// TwinCAT 3 PLC project plc01
// ProgramVersion: 3.1.4026.20
// libraries:
//   Tc2_Standard, * (Beckhoff Automation GmbH)
//   Tc2_System, * (Beckhoff Automation GmbH)
//   Tc2_Utilities, * (Beckhoff Automation GmbH)
//   Tc3_Event, * (www.peterzerlauth.com)
// project tree:
//   / FastTask.TcTTO (not stored), PlcTask.TcTTO (not stored)
//   POUs/ FAST.TcPOU (not stored), FB_TestSlow.TcPOU, FB_TestFast.TcPOU, MAIN.TcPOU
// real-time tasks:
//   TASK SlowTask: cycle T#20ms, priority 20, ADS port 350
//   TASK FastTask: cycle T#1ms, priority 1, ADS port 351

// ---- POUs/FB_TestSlow.TcPOU
FUNCTION_BLOCK FB_TestSlow
VAR_INPUT
END_VAR
VAR_OUTPUT
END_VAR
VAR
	fbEvent: 			Tc3_Event.FB_Event;
	bVerbose:			BOOL;
	bInfo:				BOOL;
	bWarning:			BOOL;
	bError:				BOOL;
	bCritical:			BOOL;

END_VAR

fbEvent();

// Demonstration of FB_Event usage with various log levels and argument types

IF bVerbose THEN
	fbEvent.P_Argument.M_AddINT(134052566194980000);
	fbEvent.P_Argument.M_AddSTRING('mm');
	fbEvent.M_Verbose('V message %s %s');
END_IF

IF bInfo THEN
	fbEvent.P_Argument.M_AddREAL(33.134581234, 3);
	fbEvent.P_Argument.M_AddSTRING('mm');
	fbEvent.M_Info('I message %s %s', 0);
END_IF

IF bWarning THEN
	fbEvent.M_Warning('W message', 0);
	fbEvent.M_Warning('B message', 475719253);
END_IF

IF bError THEN
	fbEvent.M_Error('E message', 475719235);
END_IF

IF bCritical THEN
	fbEvent.M_Error('Input %s is simulated', 849363082);
END_IF

PROPERTY PUBLIC P_Event : reference to FB_event
GET
P_Event ref= fbEvent;
END_GET
END_PROPERTY

END_FUNCTION_BLOCK

// ---- POUs/FB_TestFast.TcPOU
FUNCTION_BLOCK FB_TestFast
VAR_INPUT
END_VAR
VAR_OUTPUT
END_VAR
VAR
	fbEvent: 			Tc3_Event.FB_Event;
	bVerbose:			BOOL;
	bInfo:				BOOL;
	bWarning:			BOOL;
	bError:				BOOL;
	bCritical:			BOOL;

END_VAR

fbEvent();

// Demonstration of FB_Event usage with various log levels and argument types

IF bVerbose THEN
	fbEvent.P_Argument.M_AddINT(134052566194980000);
	fbEvent.P_Argument.M_AddSTRING('mm');
	fbEvent.M_Verbose('V message %s %s');
END_IF

IF bInfo THEN
	fbEvent.P_Argument.M_AddREAL(33.134581234, 3);
	fbEvent.P_Argument.M_AddSTRING('mm');
	fbEvent.M_Info('I message %s %s', 828536003);
END_IF

IF bWarning THEN
	fbEvent.M_Warning('W message', 475719253);
	fbEvent.M_Warning('W message', 475719253);
END_IF

IF bError THEN
	fbEvent.M_Error('E message', 475719235);
END_IF

IF bCritical THEN
	fbEvent.M_Critical('C message', 475719233); ///839384782
	fbEvent.M_Critical('B message', 0); 
END_IF

PROPERTY PUBLIC P_Event : reference to FB_event
GET
P_Event ref= fbEvent;
END_GET
END_PROPERTY

END_FUNCTION_BLOCK

// ---- POUs/MAIN.TcPOU
PROGRAM MAIN
VAR
	fbLogger:			Tc3_Event.FB_LoggerManager;
	fbHmiLogger:		Tc3_Event.FB_HmiLogger;
	fbFileLogger:		Tc3_Event.FB_FileLogger;
	fbTcLogger:			Tc3_Event.FB_TcLogger;
	fbTest:				FB_TestSlow;
  	exception:			__SYSTEM.ExceptionCode;	
	bReset: BOOL;
END_VAR

__TRY
	IF exception = __SYSTEM.ExceptionCode.RTSEXCPT_NOEXCEPTION THEN
		fbLogger.M_Add(fbHmiLogger);
		fbLogger.M_Add(fbFileLogger);
			
		fbHmiLogger();
		fbFileLogger.sPathName:= 'C:\temp\log.txt';
		fbFileLogger();

		
		
		IF bReset THEN
			fbTest.P_Event.M_Reset();
		END_IF
		
		fbTest.P_Event.P_Logger:= fbLogger;
		
		fbTest();	
		
// 		fbTest1000.P_Event.P_Logger:= fbLogger;
// 		fbTest1000();
		
	END_IF

__CATCH(exception)

__ENDTRY

END_PROGRAM
